// TIA Portal V17 export
// export: Created 2024-08-26T21:10:47.941698Z, ExportSetting WithDefaults, DisplayName Totally Integrated Automation Portal, DisplayVersion V17 Update 7, DisplayName TIA Portal Openness, DisplayVersion V17 Update 7, DisplayName TIA Portal Version Control Interface, DisplayVersion V17, DisplayName SINAMICS Startdrive Advanced, DisplayVersion V17 SP2, DisplayName SINAMICS Startdrive G110M, G120, G120C, G120D, G120P, G115D, DisplayVersion V17 SP2, DisplayName SINAMICS Startdrive G130, G150, S120, S150, SINAMICS MV, S210, DisplayVersion V17 SP2, DisplayName STEP 7 Professional, DisplayVersion V17 Update 7, DisplayName STEP 7 Safety, DisplayVersion V17 Update 6, DisplayName WinCC Advanced / Unified PC, DisplayVersion V17 Update 7
FUNCTION "inputsMapping" : Void   // FC1, LAD
{ S7_Optimized_Access := 'TRUE' }
VERSION : 0.1
// stored: AutoNumber true, IsIECCheckEnabled false, SetENOAutomatically false, UDAEnableTagReadback false
BEGIN

REGION Network 1: A00.- CLEAR DATA
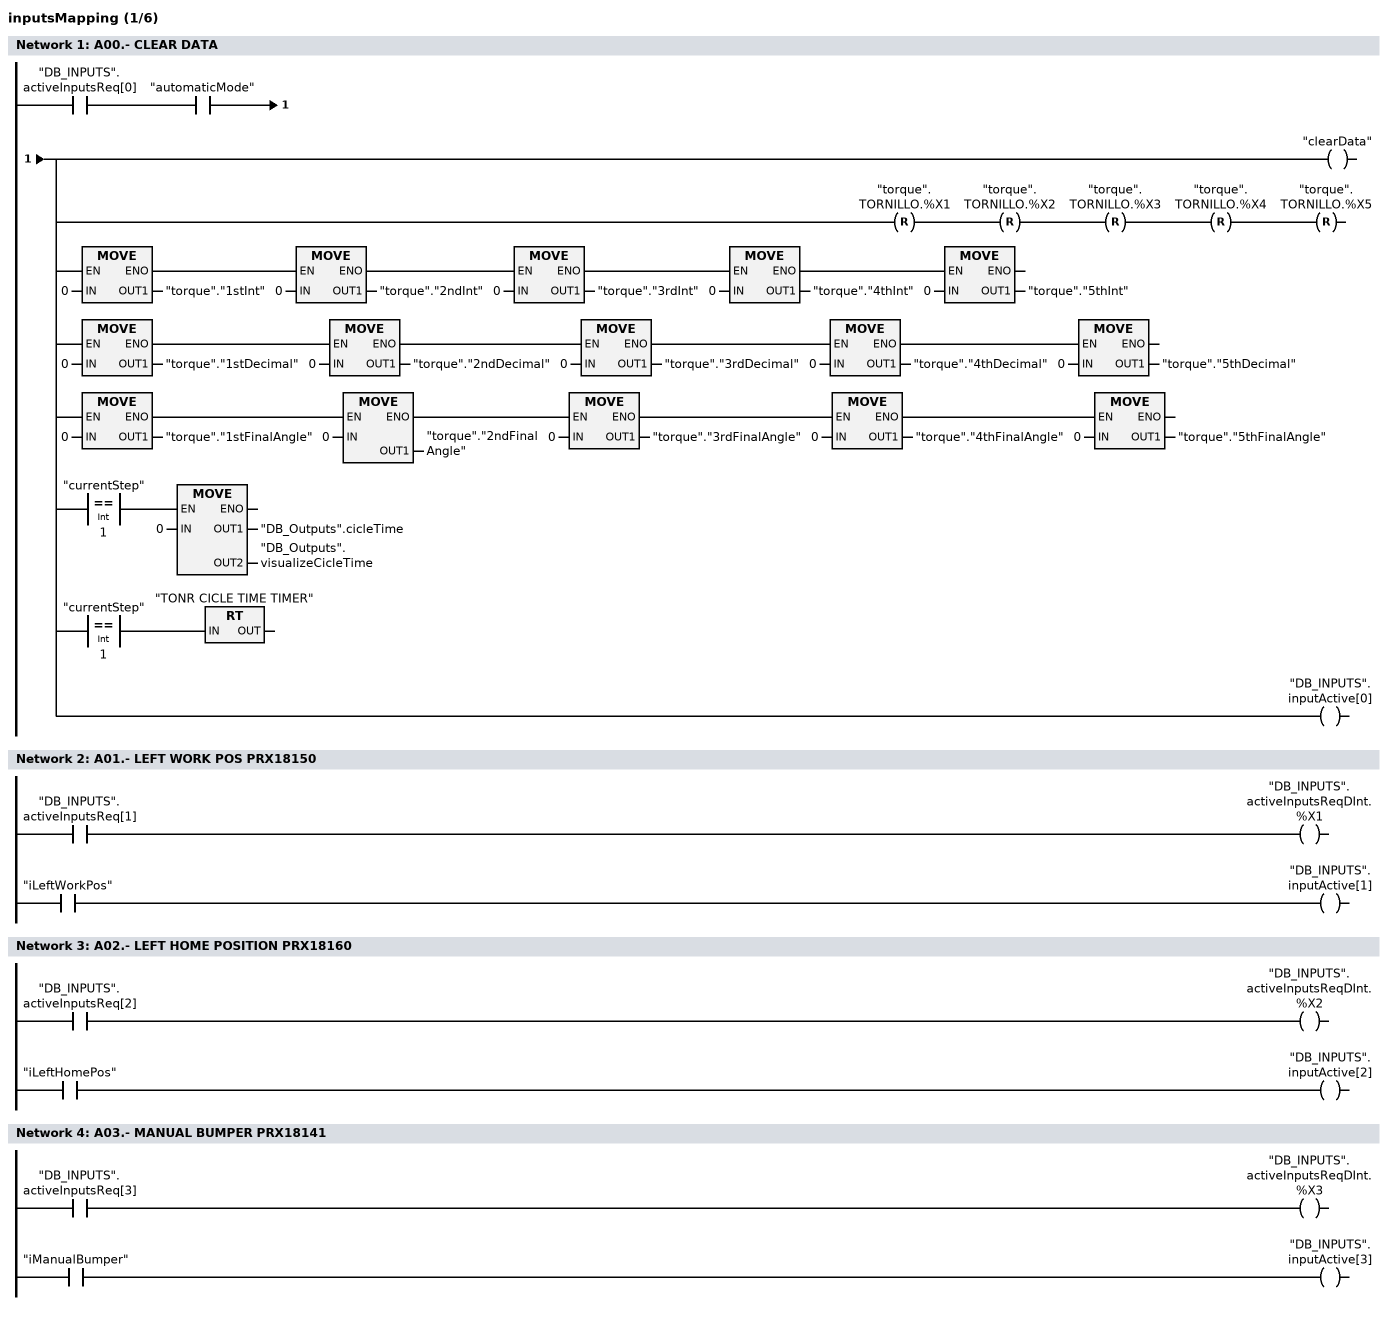
   RUNG wire#powerrail
      Contact( "DB_INPUTS".activeInputsReq[0] )
      Contact( "automaticMode" )
      wire#w1
      Coil( "clearData" )
   END_RUNG
   RUNG wire#w1
      R_Coil( "torque".TORNILLO.%X1 )
      R_Coil( "torque".TORNILLO.%X2 )
      R_Coil( "torque".TORNILLO.%X3 )
      R_Coil( "torque".TORNILLO.%X4 )
      R_Coil( "torque".TORNILLO.%X5 )
   END_RUNG
   RUNG wire#w1
      Move(in := 0, out1 => "torque"."1stInt")
      Move(in := 0, out1 => "torque"."2ndInt")
      Move(in := 0, out1 => "torque"."3rdInt")
      Move(in := 0, out1 => "torque"."4thInt")
      Move(in := 0, out1 => "torque"."5thInt")
   END_RUNG
   RUNG wire#w1
      Move(in := 0, out1 => "torque"."1stDecimal")
      Move(in := 0, out1 => "torque"."2ndDecimal")
      Move(in := 0, out1 => "torque"."3rdDecimal")
      Move(in := 0, out1 => "torque"."4thDecimal")
      Move(in := 0, out1 => "torque"."5thDecimal")
   END_RUNG
   RUNG wire#w1
      Move(in := 0, out1 => "torque"."1stFinalAngle")
      Move(in := 0, out1 => "torque"."2ndFinalAngle")
      Move(in := 0, out1 => "torque"."3rdFinalAngle")
      Move(in := 0, out1 => "torque"."4thFinalAngle")
      Move(in := 0, out1 => "torque"."5thFinalAngle")
   END_RUNG
   RUNG wire#w1
      { S7_Templates := "SrcType := Int" } EQ_Contact(in1 := "currentStep", in2 := 1)
      Move(in := 0, out1 => "DB_Outputs".cicleTime, out2 => "DB_Outputs".visualizeCicleTime)
   END_RUNG
   RUNG wire#w1
      { S7_Templates := "SrcType := Int" } EQ_Contact(in1 := "currentStep", in2 := 1)
      RT_Coil( "TONR CICLE TIME TIMER" )
   END_RUNG
   RUNG wire#w1
      Coil( "DB_INPUTS".inputActive[0] )
   END_RUNG
   // the same network as SCL:
   "clearData" := "DB_INPUTS".activeInputsReq[0] AND "automaticMode";
   IF "clearData" THEN
       "torque".TORNILLO.%X1 := FALSE;
       "torque".TORNILLO.%X2 := FALSE;
       "torque".TORNILLO.%X3 := FALSE;
       "torque".TORNILLO.%X4 := FALSE;
       "torque".TORNILLO.%X5 := FALSE;
       "torque"."1stInt" := 0;
       "torque"."2ndInt" := 0;
       "torque"."3rdInt" := 0;
       "torque"."4thInt" := 0;
       "torque"."5thInt" := 0;
       "torque"."1stDecimal" := 0;
       "torque"."2ndDecimal" := 0;
       "torque"."3rdDecimal" := 0;
       "torque"."4thDecimal" := 0;
       "torque"."5thDecimal" := 0;
       "torque"."1stFinalAngle" := 0;
       "torque"."2ndFinalAngle" := 0;
       "torque"."3rdFinalAngle" := 0;
       "torque"."4thFinalAngle" := 0;
       "torque"."5thFinalAngle" := 0;
   END_IF;
   IF "clearData" AND ("currentStep" = 1) THEN
       "DB_Outputs".cicleTime := 0;
       "DB_Outputs".visualizeCicleTime := 0;
       RESET_TIMER("TONR CICLE TIME TIMER");
   END_IF;
   "DB_INPUTS".inputActive[0] := "clearData";
END_REGION

REGION Network 2: A01.- LEFT WORK POS PRX18150
   RUNG wire#powerrail
      Contact( "DB_INPUTS".activeInputsReq[1] )
      Coil( "DB_INPUTS".activeInputsReqDInt.%X1 )
   END_RUNG
   RUNG wire#powerrail
      Contact( "iLeftWorkPos" )
      Coil( "DB_INPUTS".inputActive[1] )
   END_RUNG
   // the same network as SCL:
   "DB_INPUTS".activeInputsReqDInt.%X1 := "DB_INPUTS".activeInputsReq[1];
   "DB_INPUTS".inputActive[1] := "iLeftWorkPos";
END_REGION

REGION Network 3: A02.- LEFT HOME POSITION PRX18160
   RUNG wire#powerrail
      Contact( "DB_INPUTS".activeInputsReq[2] )
      Coil( "DB_INPUTS".activeInputsReqDInt.%X2 )
   END_RUNG
   RUNG wire#powerrail
      Contact( "iLeftHomePos" )
      Coil( "DB_INPUTS".inputActive[2] )
   END_RUNG
   // the same network as SCL:
   "DB_INPUTS".activeInputsReqDInt.%X2 := "DB_INPUTS".activeInputsReq[2];
   "DB_INPUTS".inputActive[2] := "iLeftHomePos";
END_REGION

REGION Network 4: A03.- MANUAL BUMPER PRX18141
   RUNG wire#powerrail
      Contact( "DB_INPUTS".activeInputsReq[3] )
      Coil( "DB_INPUTS".activeInputsReqDInt.%X3 )
   END_RUNG
   RUNG wire#powerrail
      Contact( "iManualBumper" )
      Coil( "DB_INPUTS".inputActive[3] )
   END_RUNG
   // the same network as SCL:
   "DB_INPUTS".activeInputsReqDInt.%X3 := "DB_INPUTS".activeInputsReq[3];
   "DB_INPUTS".inputActive[3] := "iManualBumper";
END_REGION

REGION Network 5: A04.- LEFT MANUAL TOOLING EXT OK PRX18151
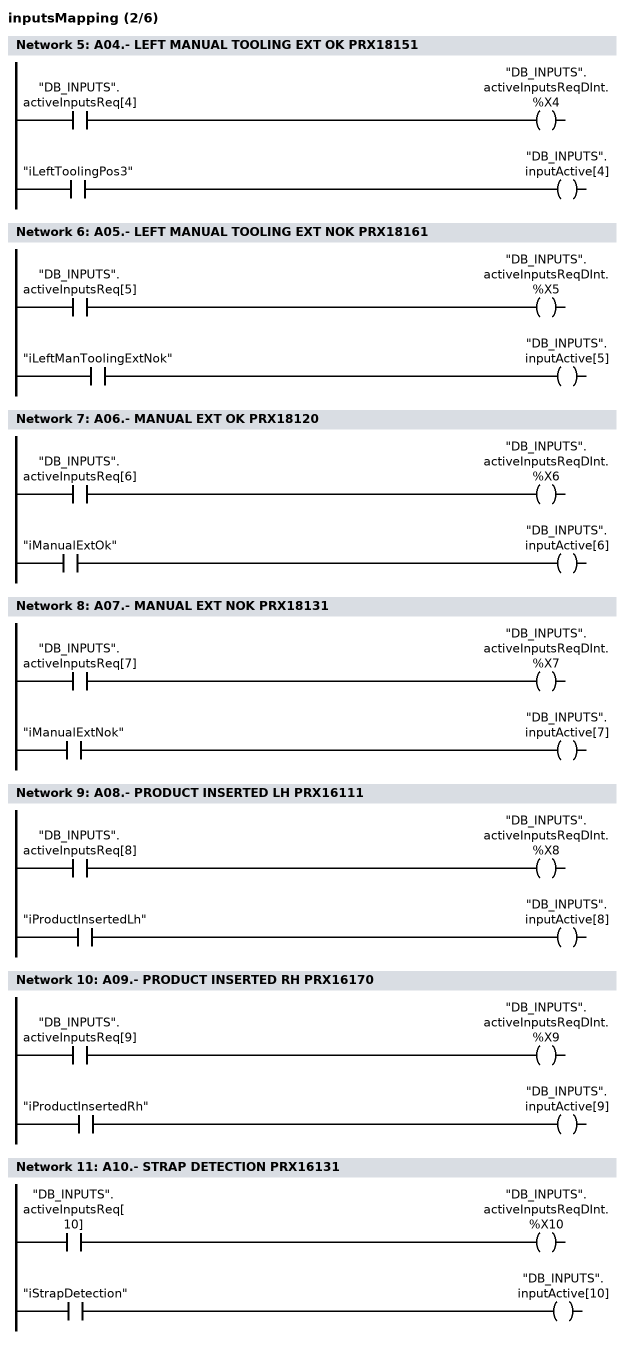
   RUNG wire#powerrail
      Contact( "DB_INPUTS".activeInputsReq[4] )
      Coil( "DB_INPUTS".activeInputsReqDInt.%X4 )
   END_RUNG
   RUNG wire#powerrail
      Contact( "iLeftToolingPos3" )
      Coil( "DB_INPUTS".inputActive[4] )
   END_RUNG
   // the same network as SCL:
   "DB_INPUTS".activeInputsReqDInt.%X4 := "DB_INPUTS".activeInputsReq[4];
   "DB_INPUTS".inputActive[4] := "iLeftToolingPos3";
END_REGION

REGION Network 6: A05.- LEFT MANUAL TOOLING EXT NOK PRX18161
   RUNG wire#powerrail
      Contact( "DB_INPUTS".activeInputsReq[5] )
      Coil( "DB_INPUTS".activeInputsReqDInt.%X5 )
   END_RUNG
   RUNG wire#powerrail
      Contact( "iLeftManToolingExtNok" )
      Coil( "DB_INPUTS".inputActive[5] )
   END_RUNG
   // the same network as SCL:
   "DB_INPUTS".activeInputsReqDInt.%X5 := "DB_INPUTS".activeInputsReq[5];
   "DB_INPUTS".inputActive[5] := "iLeftManToolingExtNok";
END_REGION

REGION Network 7: A06.- MANUAL EXT OK PRX18120
   RUNG wire#powerrail
      Contact( "DB_INPUTS".activeInputsReq[6] )
      Coil( "DB_INPUTS".activeInputsReqDInt.%X6 )
   END_RUNG
   RUNG wire#powerrail
      Contact( "iManualExtOk" )
      Coil( "DB_INPUTS".inputActive[6] )
   END_RUNG
   // the same network as SCL:
   "DB_INPUTS".activeInputsReqDInt.%X6 := "DB_INPUTS".activeInputsReq[6];
   "DB_INPUTS".inputActive[6] := "iManualExtOk";
END_REGION

REGION Network 8: A07.- MANUAL EXT NOK PRX18131
   RUNG wire#powerrail
      Contact( "DB_INPUTS".activeInputsReq[7] )
      Coil( "DB_INPUTS".activeInputsReqDInt.%X7 )
   END_RUNG
   RUNG wire#powerrail
      Contact( "iManualExtNok" )
      Coil( "DB_INPUTS".inputActive[7] )
   END_RUNG
   // the same network as SCL:
   "DB_INPUTS".activeInputsReqDInt.%X7 := "DB_INPUTS".activeInputsReq[7];
   "DB_INPUTS".inputActive[7] := "iManualExtNok";
END_REGION

REGION Network 9: A08.- PRODUCT INSERTED LH PRX16111
   RUNG wire#powerrail
      Contact( "DB_INPUTS".activeInputsReq[8] )
      Coil( "DB_INPUTS".activeInputsReqDInt.%X8 )
   END_RUNG
   RUNG wire#powerrail
      Contact( "iProductInsertedLh" )
      Coil( "DB_INPUTS".inputActive[8] )
   END_RUNG
   // the same network as SCL:
   "DB_INPUTS".activeInputsReqDInt.%X8 := "DB_INPUTS".activeInputsReq[8];
   "DB_INPUTS".inputActive[8] := "iProductInsertedLh";
END_REGION

REGION Network 10: A09.- PRODUCT INSERTED RH PRX16170
   RUNG wire#powerrail
      Contact( "DB_INPUTS".activeInputsReq[9] )
      Coil( "DB_INPUTS".activeInputsReqDInt.%X9 )
   END_RUNG
   RUNG wire#powerrail
      Contact( "iProductInsertedRh" )
      Coil( "DB_INPUTS".inputActive[9] )
   END_RUNG
   // the same network as SCL:
   "DB_INPUTS".activeInputsReqDInt.%X9 := "DB_INPUTS".activeInputsReq[9];
   "DB_INPUTS".inputActive[9] := "iProductInsertedRh";
END_REGION

REGION Network 11: A10.- STRAP DETECTION PRX16131
   RUNG wire#powerrail
      Contact( "DB_INPUTS".activeInputsReq[10] )
      Coil( "DB_INPUTS".activeInputsReqDInt.%X10 )
   END_RUNG
   RUNG wire#powerrail
      Contact( "iStrapDetection" )
      Coil( "DB_INPUTS".inputActive[10] )
   END_RUNG
   // the same network as SCL:
   "DB_INPUTS".activeInputsReqDInt.%X10 := "DB_INPUTS".activeInputsReq[10];
   "DB_INPUTS".inputActive[10] := "iStrapDetection";
END_REGION

REGION Network 12: A11.- PRESENT LEFT MANUAL FRAME PRX17111
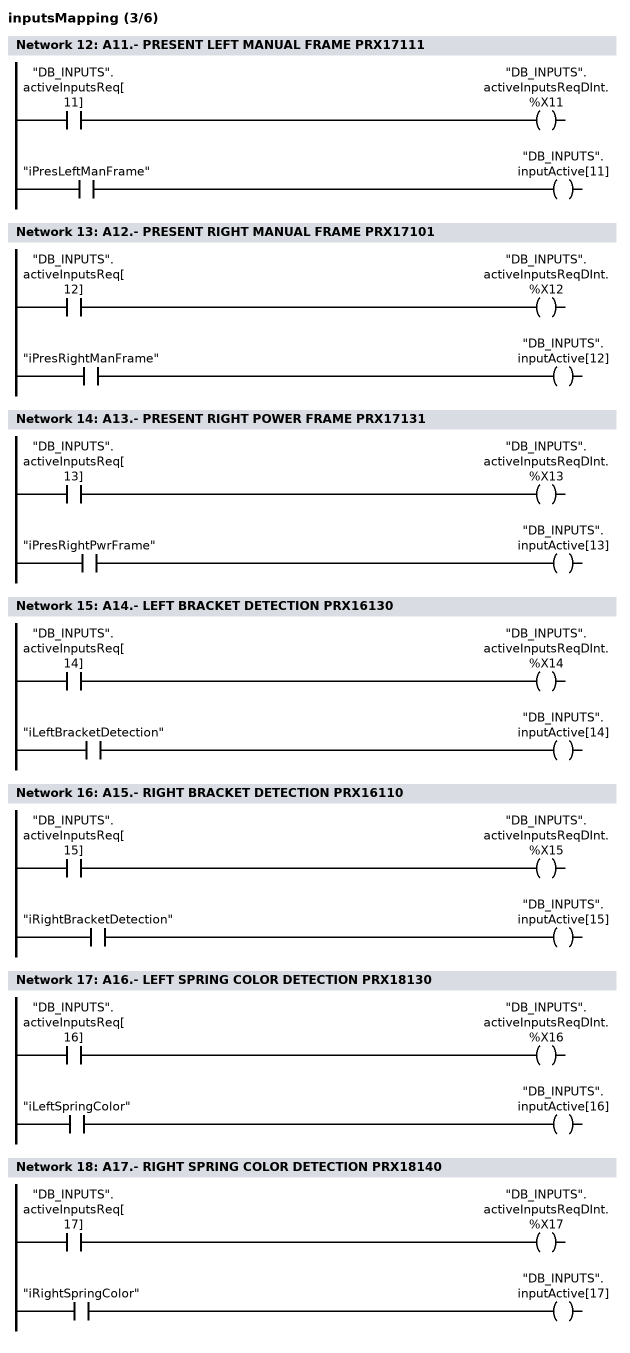
   RUNG wire#powerrail
      Contact( "DB_INPUTS".activeInputsReq[11] )
      Coil( "DB_INPUTS".activeInputsReqDInt.%X11 )
   END_RUNG
   RUNG wire#powerrail
      Contact( "iPresLeftManFrame" )
      Coil( "DB_INPUTS".inputActive[11] )
   END_RUNG
   // the same network as SCL:
   "DB_INPUTS".activeInputsReqDInt.%X11 := "DB_INPUTS".activeInputsReq[11];
   "DB_INPUTS".inputActive[11] := "iPresLeftManFrame";
END_REGION

REGION Network 13: A12.- PRESENT RIGHT MANUAL FRAME PRX17101
   RUNG wire#powerrail
      Contact( "DB_INPUTS".activeInputsReq[12] )
      Coil( "DB_INPUTS".activeInputsReqDInt.%X12 )
   END_RUNG
   RUNG wire#powerrail
      Contact( "iPresRightManFrame" )
      Coil( "DB_INPUTS".inputActive[12] )
   END_RUNG
   // the same network as SCL:
   "DB_INPUTS".activeInputsReqDInt.%X12 := "DB_INPUTS".activeInputsReq[12];
   "DB_INPUTS".inputActive[12] := "iPresRightManFrame";
END_REGION

REGION Network 14: A13.- PRESENT RIGHT POWER FRAME PRX17131
   RUNG wire#powerrail
      Contact( "DB_INPUTS".activeInputsReq[13] )
      Coil( "DB_INPUTS".activeInputsReqDInt.%X13 )
   END_RUNG
   RUNG wire#powerrail
      Contact( "iPresRightPwrFrame" )
      Coil( "DB_INPUTS".inputActive[13] )
   END_RUNG
   // the same network as SCL:
   "DB_INPUTS".activeInputsReqDInt.%X13 := "DB_INPUTS".activeInputsReq[13];
   "DB_INPUTS".inputActive[13] := "iPresRightPwrFrame";
END_REGION

REGION Network 15: A14.- LEFT BRACKET DETECTION PRX16130
   RUNG wire#powerrail
      Contact( "DB_INPUTS".activeInputsReq[14] )
      Coil( "DB_INPUTS".activeInputsReqDInt.%X14 )
   END_RUNG
   RUNG wire#powerrail
      Contact( "iLeftBracketDetection" )
      Coil( "DB_INPUTS".inputActive[14] )
   END_RUNG
   // the same network as SCL:
   "DB_INPUTS".activeInputsReqDInt.%X14 := "DB_INPUTS".activeInputsReq[14];
   "DB_INPUTS".inputActive[14] := "iLeftBracketDetection";
END_REGION

REGION Network 16: A15.- RIGHT BRACKET DETECTION PRX16110
   RUNG wire#powerrail
      Contact( "DB_INPUTS".activeInputsReq[15] )
      Coil( "DB_INPUTS".activeInputsReqDInt.%X15 )
   END_RUNG
   RUNG wire#powerrail
      Contact( "iRightBracketDetection" )
      Coil( "DB_INPUTS".inputActive[15] )
   END_RUNG
   // the same network as SCL:
   "DB_INPUTS".activeInputsReqDInt.%X15 := "DB_INPUTS".activeInputsReq[15];
   "DB_INPUTS".inputActive[15] := "iRightBracketDetection";
END_REGION

REGION Network 17: A16.- LEFT SPRING COLOR DETECTION PRX18130
   RUNG wire#powerrail
      Contact( "DB_INPUTS".activeInputsReq[16] )
      Coil( "DB_INPUTS".activeInputsReqDInt.%X16 )
   END_RUNG
   RUNG wire#powerrail
      Contact( "iLeftSpringColor" )
      Coil( "DB_INPUTS".inputActive[16] )
   END_RUNG
   // the same network as SCL:
   "DB_INPUTS".activeInputsReqDInt.%X16 := "DB_INPUTS".activeInputsReq[16];
   "DB_INPUTS".inputActive[16] := "iLeftSpringColor";
END_REGION

REGION Network 18: A17.- RIGHT SPRING COLOR DETECTION PRX18140
   RUNG wire#powerrail
      Contact( "DB_INPUTS".activeInputsReq[17] )
      Coil( "DB_INPUTS".activeInputsReqDInt.%X17 )
   END_RUNG
   RUNG wire#powerrail
      Contact( "iRightSpringColor" )
      Coil( "DB_INPUTS".inputActive[17] )
   END_RUNG
   // the same network as SCL:
   "DB_INPUTS".activeInputsReqDInt.%X17 := "DB_INPUTS".activeInputsReq[17];
   "DB_INPUTS".inputActive[17] := "iRightSpringColor";
END_REGION

REGION Network 19: A18.- TORQUE TOOLING HOME PRX16151
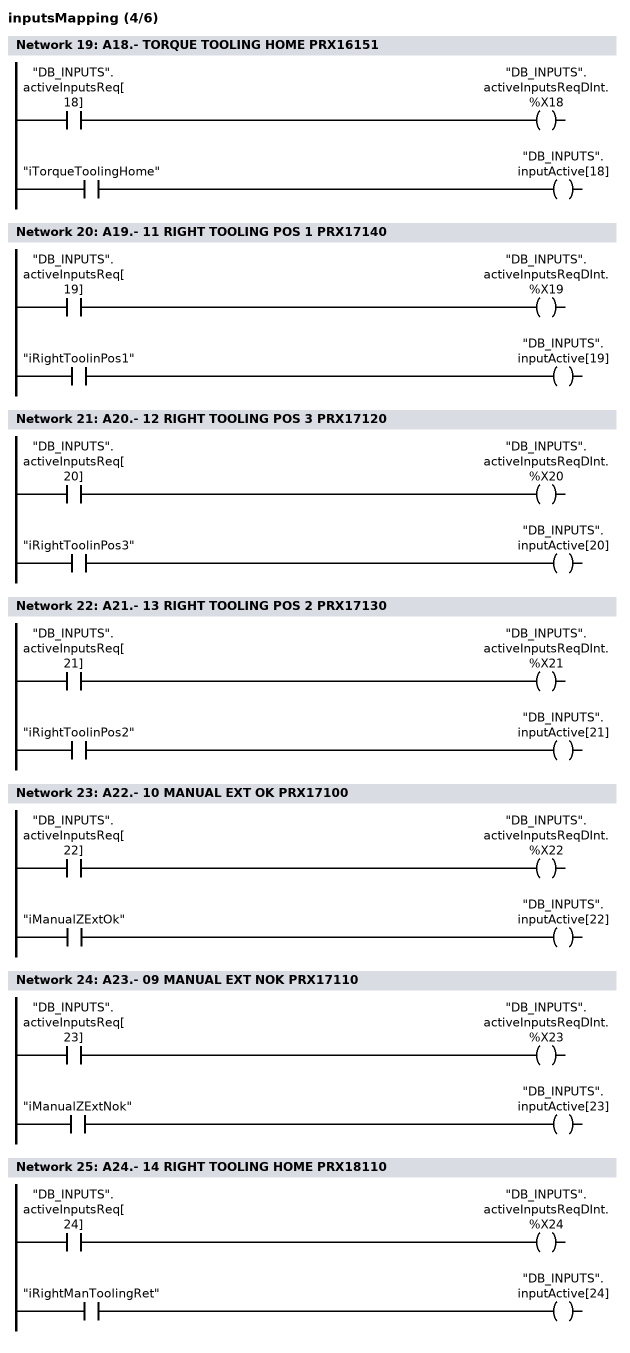
   RUNG wire#powerrail
      Contact( "DB_INPUTS".activeInputsReq[18] )
      Coil( "DB_INPUTS".activeInputsReqDInt.%X18 )
   END_RUNG
   RUNG wire#powerrail
      Contact( "iTorqueToolingHome" )
      Coil( "DB_INPUTS".inputActive[18] )
   END_RUNG
   // the same network as SCL:
   "DB_INPUTS".activeInputsReqDInt.%X18 := "DB_INPUTS".activeInputsReq[18];
   "DB_INPUTS".inputActive[18] := "iTorqueToolingHome";
END_REGION

REGION Network 20: A19.- 11 RIGHT TOOLING POS 1 PRX17140
   RUNG wire#powerrail
      Contact( "DB_INPUTS".activeInputsReq[19] )
      Coil( "DB_INPUTS".activeInputsReqDInt.%X19 )
   END_RUNG
   RUNG wire#powerrail
      Contact( "iRightToolinPos1" )
      Coil( "DB_INPUTS".inputActive[19] )
   END_RUNG
   // the same network as SCL:
   "DB_INPUTS".activeInputsReqDInt.%X19 := "DB_INPUTS".activeInputsReq[19];
   "DB_INPUTS".inputActive[19] := "iRightToolinPos1";
END_REGION

REGION Network 21: A20.- 12 RIGHT TOOLING POS 3 PRX17120
   RUNG wire#powerrail
      Contact( "DB_INPUTS".activeInputsReq[20] )
      Coil( "DB_INPUTS".activeInputsReqDInt.%X20 )
   END_RUNG
   RUNG wire#powerrail
      Contact( "iRightToolinPos3" )
      Coil( "DB_INPUTS".inputActive[20] )
   END_RUNG
   // the same network as SCL:
   "DB_INPUTS".activeInputsReqDInt.%X20 := "DB_INPUTS".activeInputsReq[20];
   "DB_INPUTS".inputActive[20] := "iRightToolinPos3";
END_REGION

REGION Network 22: A21.- 13 RIGHT TOOLING POS 2 PRX17130
   RUNG wire#powerrail
      Contact( "DB_INPUTS".activeInputsReq[21] )
      Coil( "DB_INPUTS".activeInputsReqDInt.%X21 )
   END_RUNG
   RUNG wire#powerrail
      Contact( "iRightToolinPos2" )
      Coil( "DB_INPUTS".inputActive[21] )
   END_RUNG
   // the same network as SCL:
   "DB_INPUTS".activeInputsReqDInt.%X21 := "DB_INPUTS".activeInputsReq[21];
   "DB_INPUTS".inputActive[21] := "iRightToolinPos2";
END_REGION

REGION Network 23: A22.- 10 MANUAL EXT OK PRX17100
   RUNG wire#powerrail
      Contact( "DB_INPUTS".activeInputsReq[22] )
      Coil( "DB_INPUTS".activeInputsReqDInt.%X22 )
   END_RUNG
   RUNG wire#powerrail
      Contact( "iManualZExtOk" )
      Coil( "DB_INPUTS".inputActive[22] )
   END_RUNG
   // the same network as SCL:
   "DB_INPUTS".activeInputsReqDInt.%X22 := "DB_INPUTS".activeInputsReq[22];
   "DB_INPUTS".inputActive[22] := "iManualZExtOk";
END_REGION

REGION Network 24: A23.- 09 MANUAL EXT NOK PRX17110
   RUNG wire#powerrail
      Contact( "DB_INPUTS".activeInputsReq[23] )
      Coil( "DB_INPUTS".activeInputsReqDInt.%X23 )
   END_RUNG
   RUNG wire#powerrail
      Contact( "iManualZExtNok" )
      Coil( "DB_INPUTS".inputActive[23] )
   END_RUNG
   // the same network as SCL:
   "DB_INPUTS".activeInputsReqDInt.%X23 := "DB_INPUTS".activeInputsReq[23];
   "DB_INPUTS".inputActive[23] := "iManualZExtNok";
END_REGION

REGION Network 25: A24.- 14 RIGHT TOOLING HOME PRX18110
   RUNG wire#powerrail
      Contact( "DB_INPUTS".activeInputsReq[24] )
      Coil( "DB_INPUTS".activeInputsReqDInt.%X24 )
   END_RUNG
   RUNG wire#powerrail
      Contact( "iRightManToolingRet" )
      Coil( "DB_INPUTS".inputActive[24] )
   END_RUNG
   // the same network as SCL:
   "DB_INPUTS".activeInputsReqDInt.%X24 := "DB_INPUTS".activeInputsReq[24];
   "DB_INPUTS".inputActive[24] := "iRightManToolingRet";
END_REGION

REGION Network 26: A25.- WASHER PRESENCE
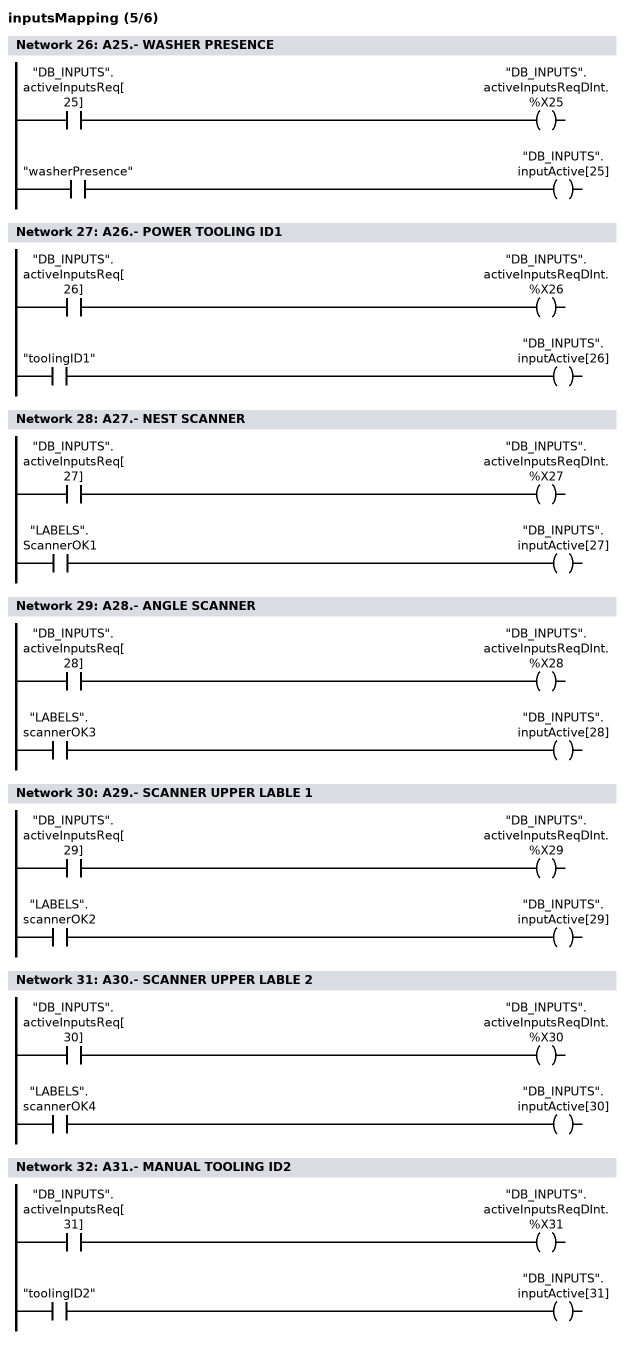
   RUNG wire#powerrail
      Contact( "DB_INPUTS".activeInputsReq[25] )
      Coil( "DB_INPUTS".activeInputsReqDInt.%X25 )
   END_RUNG
   RUNG wire#powerrail
      Contact( "washerPresence" )
      Coil( "DB_INPUTS".inputActive[25] )
   END_RUNG
   // the same network as SCL:
   "DB_INPUTS".activeInputsReqDInt.%X25 := "DB_INPUTS".activeInputsReq[25];
   "DB_INPUTS".inputActive[25] := "washerPresence";
END_REGION

REGION Network 27: A26.- POWER TOOLING ID1
   RUNG wire#powerrail
      Contact( "DB_INPUTS".activeInputsReq[26] )
      Coil( "DB_INPUTS".activeInputsReqDInt.%X26 )
   END_RUNG
   RUNG wire#powerrail
      Contact( "toolingID1" )
      Coil( "DB_INPUTS".inputActive[26] )
   END_RUNG
   // the same network as SCL:
   "DB_INPUTS".activeInputsReqDInt.%X26 := "DB_INPUTS".activeInputsReq[26];
   "DB_INPUTS".inputActive[26] := "toolingID1";
END_REGION

REGION Network 28: A27.- NEST SCANNER
   RUNG wire#powerrail
      Contact( "DB_INPUTS".activeInputsReq[27] )
      Coil( "DB_INPUTS".activeInputsReqDInt.%X27 )
   END_RUNG
   RUNG wire#powerrail
      Contact( "LABELS".ScannerOK1 )
      Coil( "DB_INPUTS".inputActive[27] )
   END_RUNG
   // the same network as SCL:
   "DB_INPUTS".activeInputsReqDInt.%X27 := "DB_INPUTS".activeInputsReq[27];
   "DB_INPUTS".inputActive[27] := "LABELS".ScannerOK1;
END_REGION

REGION Network 29: A28.- ANGLE SCANNER
   RUNG wire#powerrail
      Contact( "DB_INPUTS".activeInputsReq[28] )
      Coil( "DB_INPUTS".activeInputsReqDInt.%X28 )
   END_RUNG
   RUNG wire#powerrail
      Contact( "LABELS".scannerOK3 )
      Coil( "DB_INPUTS".inputActive[28] )
   END_RUNG
   // the same network as SCL:
   "DB_INPUTS".activeInputsReqDInt.%X28 := "DB_INPUTS".activeInputsReq[28];
   "DB_INPUTS".inputActive[28] := "LABELS".scannerOK3;
END_REGION

REGION Network 30: A29.- SCANNER UPPER LABLE 1
   RUNG wire#powerrail
      Contact( "DB_INPUTS".activeInputsReq[29] )
      Coil( "DB_INPUTS".activeInputsReqDInt.%X29 )
   END_RUNG
   RUNG wire#powerrail
      Contact( "LABELS".scannerOK2 )
      Coil( "DB_INPUTS".inputActive[29] )
   END_RUNG
   // the same network as SCL:
   "DB_INPUTS".activeInputsReqDInt.%X29 := "DB_INPUTS".activeInputsReq[29];
   "DB_INPUTS".inputActive[29] := "LABELS".scannerOK2;
END_REGION

REGION Network 31: A30.- SCANNER UPPER LABLE 2
   RUNG wire#powerrail
      Contact( "DB_INPUTS".activeInputsReq[30] )
      Coil( "DB_INPUTS".activeInputsReqDInt.%X30 )
   END_RUNG
   RUNG wire#powerrail
      Contact( "LABELS".scannerOK4 )
      Coil( "DB_INPUTS".inputActive[30] )
   END_RUNG
   // the same network as SCL:
   "DB_INPUTS".activeInputsReqDInt.%X30 := "DB_INPUTS".activeInputsReq[30];
   "DB_INPUTS".inputActive[30] := "LABELS".scannerOK4;
END_REGION

REGION Network 32: A31.- MANUAL TOOLING ID2
   RUNG wire#powerrail
      Contact( "DB_INPUTS".activeInputsReq[31] )
      Coil( "DB_INPUTS".activeInputsReqDInt.%X31 )
   END_RUNG
   RUNG wire#powerrail
      Contact( "toolingID2" )
      Coil( "DB_INPUTS".inputActive[31] )
   END_RUNG
   // the same network as SCL:
   "DB_INPUTS".activeInputsReqDInt.%X31 := "DB_INPUTS".activeInputsReq[31];
   "DB_INPUTS".inputActive[31] := "toolingID2";
END_REGION

REGION Network 33: HMI SENSOR OVERVIEW
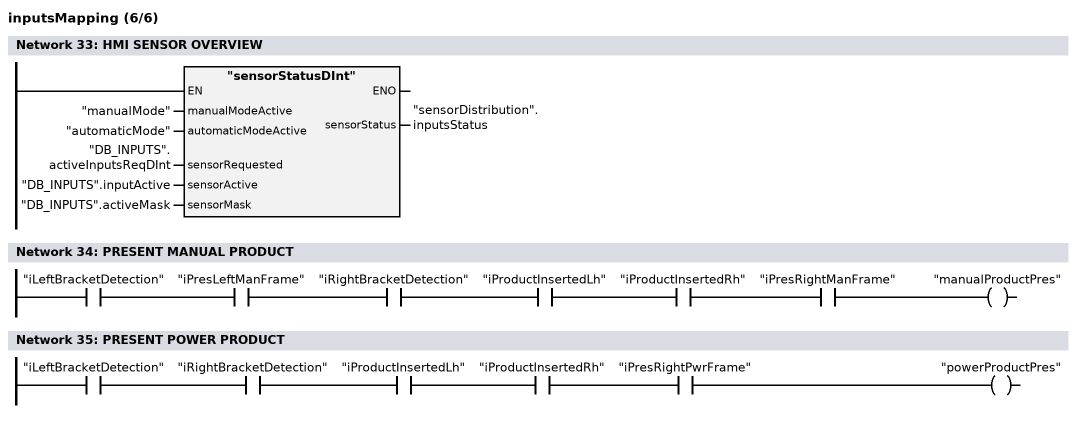
   RUNG wire#powerrail
      "sensorStatusDInt"(manualModeActive := "manualMode", automaticModeActive := "automaticMode", sensorRequested := "DB_INPUTS".activeInputsReqDInt, sensorActive := "DB_INPUTS".inputActive, sensorMask := "DB_INPUTS".activeMask, sensorStatus => "sensorDistribution".inputsStatus)
   END_RUNG
   // the same network as SCL:
   "sensorStatusDInt"(manualModeActive := "manualMode",
                      automaticModeActive := "automaticMode",
                      sensorRequested := "DB_INPUTS".activeInputsReqDInt,
                      sensorActive := "DB_INPUTS".inputActive,
                      sensorMask := "DB_INPUTS".activeMask,
                      sensorStatus => "sensorDistribution".inputsStatus);
END_REGION

REGION Network 34: PRESENT MANUAL PRODUCT
   RUNG wire#powerrail
      Contact( "iLeftBracketDetection" )
      Contact( "iPresLeftManFrame" )
      Contact( "iRightBracketDetection" )
      Contact( "iProductInsertedLh" )
      Contact( "iProductInsertedRh" )
      Contact( "iPresRightManFrame" )
      Coil( "manualProductPres" )
   END_RUNG
   // the same network as SCL:
   "manualProductPres" := "iLeftBracketDetection" AND "iPresLeftManFrame" AND "iRightBracketDetection" AND "iProductInsertedLh" AND "iProductInsertedRh" AND "iPresRightManFrame";
END_REGION

REGION Network 35: PRESENT POWER PRODUCT
   RUNG wire#powerrail
      Contact( "iLeftBracketDetection" )
      Contact( "iRightBracketDetection" )
      Contact( "iProductInsertedLh" )
      Contact( "iProductInsertedRh" )
      Contact( "iPresRightPwrFrame" )
      Coil( "powerProductPres" )
   END_RUNG
   // the same network as SCL:
   "powerProductPres" := "iLeftBracketDetection" AND "iRightBracketDetection" AND "iProductInsertedLh" AND "iProductInsertedRh" AND "iPresRightPwrFrame";
END_REGION
END_FUNCTION
